TYPE ST_FromTc3Hmi EXTENDS ST_HMI_IN :
STRUCT
	// general
	eLanguage					: E_Language := E_Language.DE;
	sCurrentPage				: WSTRING;
	sSetTargetPageConfirm		: WSTRING;
	stPopup						: ST_PopUp_FromHmi;
	//stButton_CloseHmi			: ST_Button_FromHmi; //button close hmi
	stControlCounter			: ST_CounterControlIn;	
	
	// stations custom
	//astStation					: ARRAY[0..E_Station.eStation_nMaxIdx] OF ST_StationFromTc3Hmi;
END_STRUCT
END_TYPE

(* stored: Version 1.1.0.1
   DUT ST_FromTc3Hmi: Id {c88bc23c-f19b-4ab7-98ea-6260d8276c44} *)
